{attribute 'to_string'}
TYPE E_234FeedManager_States : (
	C234_FEEDMANAGER_DISABLED,
	C234_FEEDMANAGER_ENABLING
	
	, C234_FEEDMANAGER_AUTOFEED_OFF
	, C234_FEEDMANAGER_AUTOFEED_ON
	, C234_FEEDMANAGER_TEST_TOGGLE_HAS_DOOR
	
	, C234_FEEDMANAGER_EXTERNAL
	, C234_FEEDMANAGER_EXTERNAL_RAISE_CROSS_FEED_FENCE_AND_TRANSFER_HEIGHT_CYLS
	, C234_FEEDMANAGER_EXTERNAL_LOWER_CROSS_FEED_FENCE_AND_TRANSFER_HEIGHT_CYLS
	
	, C234_FEEDMANAGER_JOG_LOWER_CROSS_FEED_FENCE_AND_TRANSFER_HEIGHT_CYLS
	, C234_FEEDMANAGER_INLINE_JOGGING
	
	, C234_FEEDMANAGER_JOG_RAISE_CROSS_FEED_FENCE_AND_TRANSFER_HEIGHT_CYLS
	, C234_FEEDMANAGER_CROSS_JOGGING
	
	, C234_FEEDMANAGER_JOG_RAISE_CROSS_FEED_FENCE_AND_LOWER_TRANSFER_HEIGHT_CYLS
	, C234_FEEDMANAGER_TO_FENCE_JOGGING
	
	, C234_FEEDMANAGER_ROTATE_LOWER_CROSS_FEED_FENCE_AND_TRANSFER_HEIGHT_CYLS
	, C234_FEEDMANAGER_ROTATE
	
	, C234_FEEDMANAGER_SELF_CENTER_LOWER_CROSS_FEED_FENCE_AND_TRANSFER_HEIGHT_CYLS
	, C234_FEEDMANAGER_SELF_CENTER
	
	, C234_FEEDMANAGER_INIT_START
	, C234_FEEDMANAGER_INIT_RAISE_CROSS_FEED_FENCE_AND_TRANSFER_HEIGHT_CYLS
	, C234_FEEDMANAGER_INIT_START_MOTOR
	, C234_FEEDMANAGER_INIT_FIND_C_OR_D_EYE_FALLING_EDGE
	, C234_FEEDMANAGER_INIT_STOP_MOTOR
	, C234_FEEDMANAGER_INIT_WAIT_FOR_ALL_CONVEYORS_INIT_COMPLETE
	
	, C234_FEEDMANAGER_FEEDIN_START
	, C234_FEEDMANAGER_FEEDIN_LOWER_CROSS_FEED_FENCE_AND_TRANSFER_HEIGHT_CYLS
	, C234_FEEDMANAGER_FEEDIN_REV_START_MOTOR
	, C234_FEEDMANAGER_FEEDIN_REV_FIND_RISING_EDGE_OF_INFEED_EYE
	, C234_FEEDMANAGER_FEEDIN_STOP
	, C234_FEEDMANAGER_FEEDIN_FWD_START_MOTOR
	, C234_FEEDMANAGER_FEEDIN_FIND_INFEED_EYE_FALLING_OR_DOORSTOP1_RISING
	, C234_FEEDMANAGER_FEEDIN_DOORSTOP1_RISING
	, C234_FEEDMANAGER_FEEDIN_DOORSTOP3_RISING
	, C234_FEEDMANAGER_FEEDIN_IN_MACHINE_EYE_FALLING
	, C234_FEEDMANAGER_FEEDIN_STOP_FINAL
	, C234_FEEDMANAGER_FEEDIN_CENTER_DOOR_PRE_ROTATE
	, C234_FEEDMANAGER_FEEDIN_ROTATE_DOOR
	, C234_FEEDMANAGER_FEEDIN_COMPLETE

	, C234_FEEDMANAGER_ALIGN_START
	, C234_FEEDMANAGER_ALIGN_RAISE_CROSS_FEED_FENCE_AND_LOWER_TRANSFER_HEIGHT_CYLS
	, C234_FEEDMANAGER_ALIGN_START_MOTOR
	, C234_FEEDMANAGER_ALIGN_FIND_FENCE_DOOR_SENSE_EYE_RISING_EDGE
	, C234_FEEDMANAGER_ALIGN_WAIT_FOR_AT_FENCE_POS
	, C234_FEEDMANAGER_ALIGN_STOP_MOTOR
	, C234_FEEDMANAGER_ALIGN_LOWER_CROSS_FEED_FENCE_AND_TRANSFER_HEIGHT_CYLS
	, C234_FEEDMANAGER_ALIGN_CENTER_DOOR
	, C234_FEEDMANAGER_ALIGN_COMPLETE

	, C234_FEEDMANAGER_FEEDOUT_START
	, C234_FEEDMANAGER_FEEDOUT_RAISE_CROSS_FEED_FENCE_AND_TRANSFER_HEIGHT_CYLS
	, C234_FEEDMANAGER_FEEDOUT_LOWER_CROSS_FEED_FENCE_AND_TRANSFER_HEIGHT_CYLS
	, C234_FEEDMANAGER_FEEDOUT_START_MOTOR
	, C234_FEEDMANAGER_FEEDOUT_FIND_OUTFEED_END_DOOR_SENSE_EYE_RISING_EDGE
	, C234_FEEDMANAGER_FEEDOUT_STOP_MOTOR
	, C234_FEEDMANAGER_FEEDOUT_WAIT_FOR_OK_TO_FEEDOUT
	, C234_FEEDMANAGER_FEEDOUT_RESTART_MOTOR
	, C234_FEEDMANAGER_FEEDOUT_FIND_OUTFEED_END_DOOR_SENSE_EYE_FALLING_EDGE
	, C234_FEEDMANAGER_FEEDOUT_STOP_MOTOR_FINAL
	, C234_FEEDMANAGER_FEEDOUT_COMPLETE
	
	, C234_FEEDMANAGER_ERROR	
);
END_TYPE

(* stored: Version 1.1.0.1, ProductVersion 3.1.4024.12
   DUT E_234FeedManager_States: Id {89911762-5f47-4798-b1a5-1b2dd096be2e} *)
